Universal Robots PolyScope program: Project1pick.urp

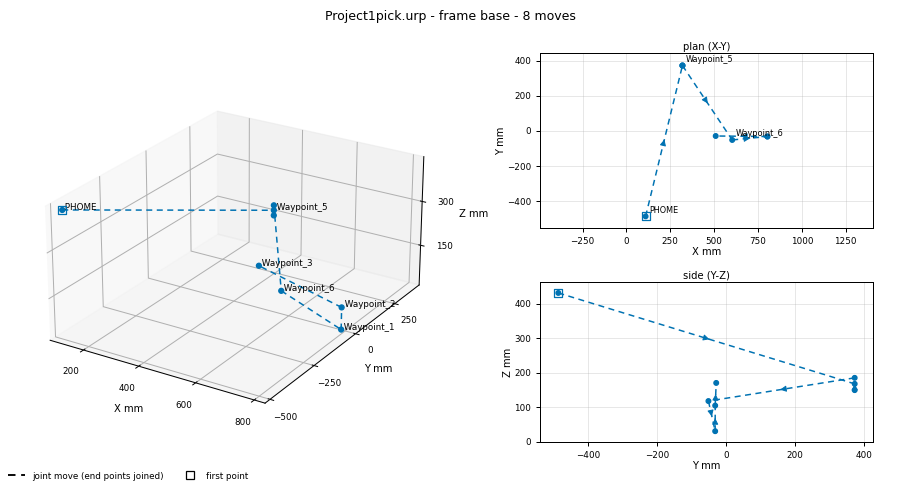
[picture p0: tool path of Project1pick.urp in frame base, 8 of 8 moves have a stored position in this frame; points joined in program order, loops and branches not executed]
Program Project1pick (installation=admin directory=/programs/TUES_530PM createdIn=3.15.8.106339 lastSavedIn=3.15.8.106339 robotSerialNumber=2015350926)
Calibrated DH parameters: a=[0, -0.425, -0.39225, 0, 0, 0]; d=[0.089159, 0, 0, 0.10915, 0.09465, 0.0823]; alpha=[1.570796, 0, 0, 1.570796, -1.570796, 0]; deltaTheta=[0, 0, 0, 0, 0, 0]
Robot Program (runOnlyOnce=true)
  Set DigitalOutput pin=digital_out[0]; digitalValue=0
  MoveJ speed 60 deg/s, acceleration 80 deg/s^2 (useActiveTCP=true)
    Waypoint PHOME: TCP in base x=109.127 y=-486.92 z=431.878 mm, rx=0.0002 ry=3.1415 rz=-0.0002 rad; joints [89.996, -90, 89.999, -90.008, -89.994, 0.002] deg
    Waypoint Waypoint_5: TCP in base x=319.215 y=373.245 z=168.003 mm, rx=0.0344 ry=3.1302 rz=0.058 rad; joints [-143.607, -78.343, 119.485, -132.91, -88.675, -232.327] deg
    Waypoint Waypoint_7: TCP in base x=319.229 y=373.19 z=149.81 mm, rx=0.0346 ry=3.1302 rz=0.058 rad; joints [-143.613, -76.428, 120.567, -135.907, -88.675, -232.327] deg
    Wait Sleep waitTime=0.5
    Set DigitalOutput pin=digital_out[0]; digitalValue=1
    Wait Sleep waitTime=0.5
    Waypoint lift: TCP in base x=319.244 y=373.173 z=185.478 mm, rx=0.0346 ry=3.13 rz=0.0581 rad; joints [-143.615, -80.067, 118.348, -130.059, -88.679, -232.329] deg
    Waypoint Waypoint_6: TCP in base x=602.972 y=-51.245 z=118.114 mm, rx=-2.1853 ry=-2.244 rz=-0.0017 rad; joints [-195.292, -60.882, 102.265, -130.946, -89.688, -196.811] deg
    Waypoint Waypoint_1: TCP in base x=803.632 y=-31.648 z=30.648 mm, rx=-2.197 ry=-2.2407 rz=-0.0051 rad; joints [-190.083, -31.326, 61.486, -120.101, -89.733, -191.212] deg
    Wait Sleep waitTime=0.5
    Set DigitalOutput pin=digital_out[0]; digitalValue=0
    Wait Sleep waitTime=0.5
    Waypoint Waypoint_2: TCP in base x=803.651 y=-31.602 z=104.99 mm, rx=-2.197 ry=-2.2409 rz=-0.0052 rad; joints [-190.079, -36.492, 59.693, -113.15, -89.733, -191.211] deg
    Waypoint Waypoint_3: TCP in base x=508.862 y=-28.636 z=170.727 mm, rx=-2.197 ry=-2.2407 rz=-0.0052 rad; joints [-195.631, -76.368, 115.777, -129.324, -89.737, -196.76] deg
